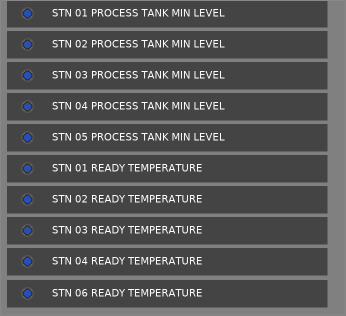
VISUALIZATION Popup_PreparationStatus  // 346x316
    Rectangle (0,0 346x316)
    Rectangle (7,0 320x27)
    Label (49,1 275x24), "STN 01 PROCESS TANK MIN LEVEL"
    Rectangle (7,31 320x27)
    Label (49,32 277x24), "STN 02 PROCESS TANK MIN LEVEL"
    Rectangle (7,62 320x27)
    Label (49,63 274x24), "STN 03 PROCESS TANK MIN LEVEL"
    Rectangle (7,93 320x27)
    Label (49,94 276x24), "STN 04 PROCESS TANK MIN LEVEL"
    Rectangle (7,124 320x27)
    Label (49,125 274x24), "STN 05 PROCESS TANK MIN LEVEL"
    Rectangle (7,155 320x27)
    Label (49,156 257x24), "STN 01 READY TEMPERATURE"
    Rectangle (7,186 320x27)
    Label (49,187 257x24), "STN 02 READY TEMPERATURE"
    Rectangle (7,217 320x27)
    Label (49,218 257x24), "STN 03 READY TEMPERATURE"
    Rectangle (7,248 320x27)
    Label (49,249 256x24), "STN 04 READY TEMPERATURE"
    Rectangle (7,280 320x27)
    Label (49,281 258x24), "STN 06 READY TEMPERATURE"
    Lamp1 (20,6 15x15), variable: ARdsMAP_HmiVariableStn[1].bProcessTankMinLevel_IND, style: Lamp-Lamp1-Blue
    Lamp1 (20,37 15x15), variable: ARdsMAP_HmiVariableStn[2].bProcessTankMinLevel_IND, style: Lamp-Lamp1-Blue
    Lamp1 (20,68 15x15), variable: ARdsMAP_HmiVariableStn[3].bProcessTankMinLevel_IND, style: Lamp-Lamp1-Blue
    Lamp1 (20,99 15x15), variable: ARdsMAP_HmiVariableStn[4].bProcessTankMinLevel_IND, style: Lamp-Lamp1-Blue
    Lamp1 (20,130 15x15), variable: ARdsMAP_HmiVariableStn[5].bProcessTankMinLevel_IND, style: Lamp-Lamp1-Blue
    Lamp1 (20,161 15x15), variable: ARbStnTempRDY[1], style: Lamp-Lamp1-Blue
    Lamp1 (20,192 15x15), variable: ARbStnTempRDY[2], style: Lamp-Lamp1-Blue
    Lamp1 (20,223 15x15), variable: ARbStnTempRDY[3], style: Lamp-Lamp1-Blue
    Lamp1 (20,254 15x15), variable: ARbStnTempRDY[4], style: Lamp-Lamp1-Blue
    Lamp1 (20,286 15x15), variable: ARbStnTempRDY[6], style: Lamp-Lamp1-Blue
END_VISUALIZATION

(* stored: Version 1.1.0.1, ProductVersion 3.1.4024.12
   Visu Popup_PreparationStatus: Id {8d59db57-fada-4d2b-8c19-de8c08ead575} *)
